{region '#Template'}
	{attribute 'Version' := '5.1.0.1'}
	{attribute 'Tags' := '"LCID": "1031", "Text": "AC, Aggregates, pre-heater, Return temperature control"'}
	{attribute 'Tags' := '"LCID": "1033", "Text": "AC, Aggregates, pre-heater, Return temperature control"'}
	{attribute 'Using' := '"Type": "Template", "URI": "BA2_Param"'}
	{attribute 'Using' := '"Type": "Template", "URI": "EC_ID"'}
	{attribute 'Description' := '"LCID": "1031", "Text": "Vorerhitzer Rücklauf Temperatur Regelung"'}
	{attribute 'Description' := '"LCID": "1033", "Text": "Pre-Heater return temperature control"'}
{endregion}
FUNCTION_BLOCK FB_BA_AC_TRtCtrl EXTENDS FB_BA_View
VAR_INPUT
	bEnPreRinse				: BOOL;
	fTRt					: REAL;
	bTWthLowLimit			: BOOL;// Außentemperatur unterer Grenzwert aktiv
	fTWth					: REAL;
	bSkipPreRinse			: BOOL; // Vorspülen überspringen // Skip pre-rinse
	bSeqActive				: BOOL;// Sequenz Regelung ist aktiv 	
END_VAR
VAR_OUTPUT
	fY						: REAL;
	bPreRinseActive			: BOOL;
	bPreRinseReady			: BOOL;
	bPreRinseDstb			: BOOL;
END_VAR
VAR_INPUT CONSTANT
	SpTRtW					: FB_BA_AV_Op;
	PreRinseDelay			: FB_BA_DlyOn;												 
	PreRinseDst				: FB_BA_BV;													   
	PreRinseSp				: FB_BA_Scale_02;																		
	Ctrl					: FB_BA_Loop;	
END_VAR
VAR
	rtrigPreRinse			: R_TRIG;
	rsPreRinseReady			: RS;
	rsPreRinseActive		: RS;
	PreRinseHys				: FB_BA_Swi2P;
END_VAR

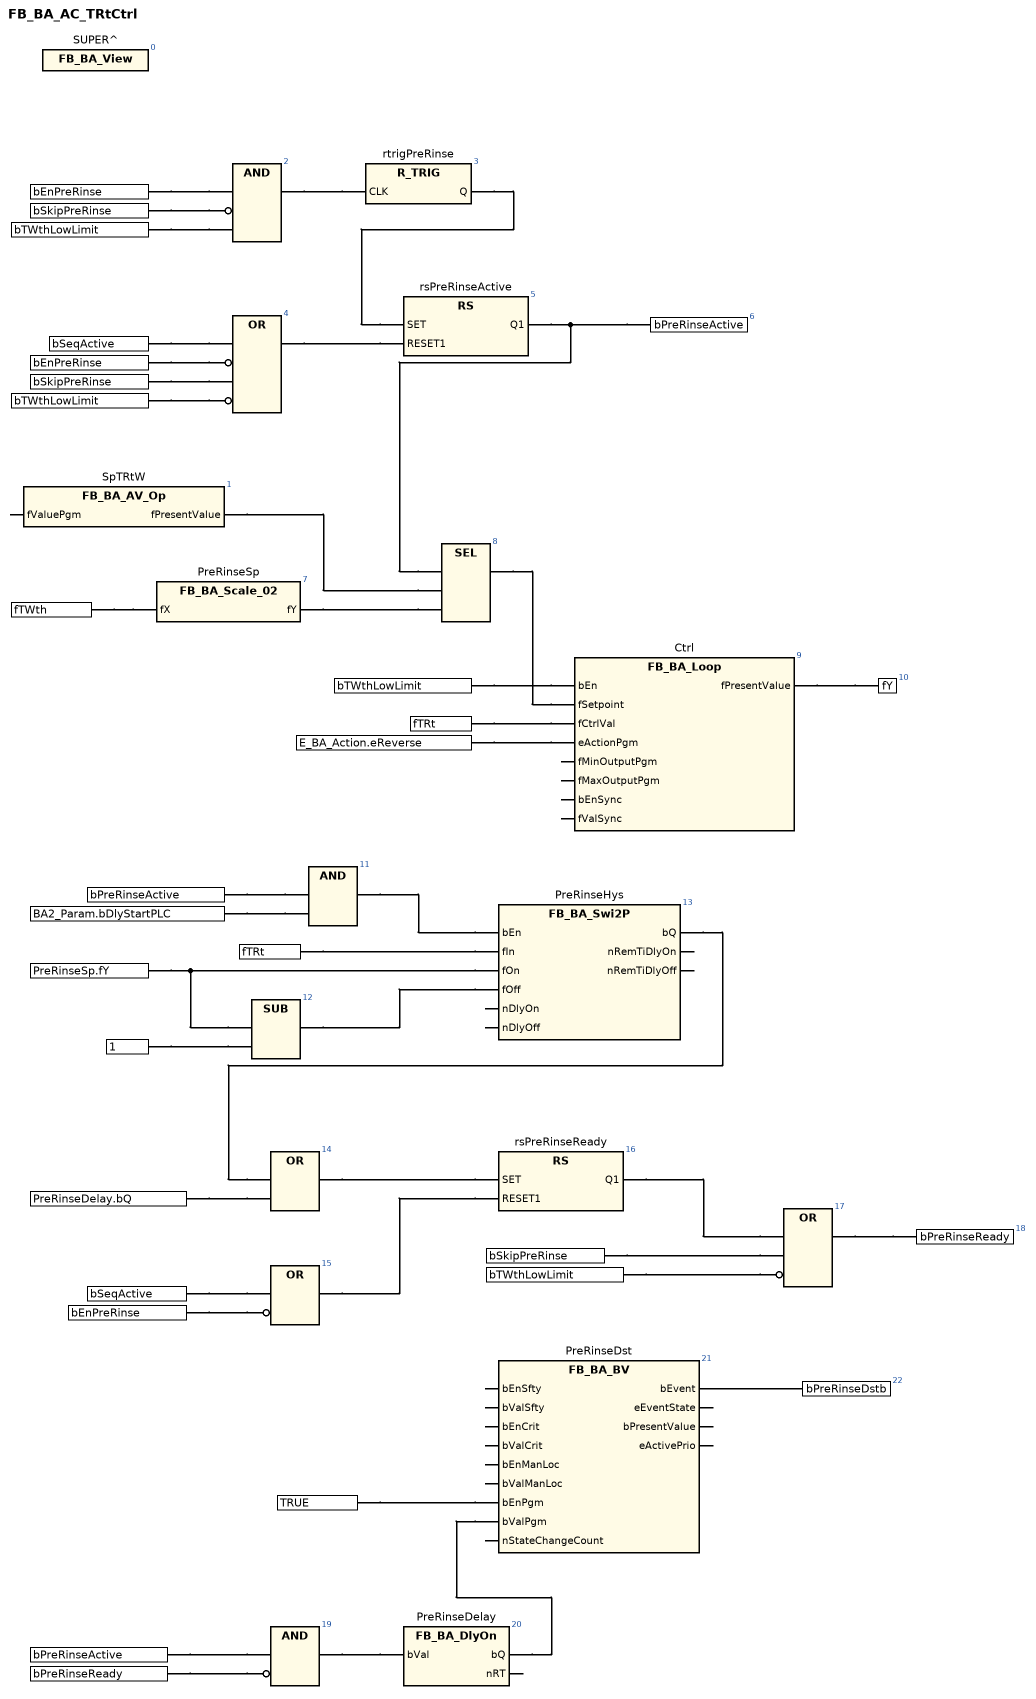
SUPER^(); // FB_BA_View
SpTRtW(); // FB_BA_AV_Op
rtrigPreRinse(CLK := bEnPreRinse AND NOT bSkipPreRinse AND bTWthLowLimit); // R_TRIG
rsPreRinseActive(SET := rtrigPreRinse.Q, RESET1 := bSeqActive OR NOT bEnPreRinse OR bSkipPreRinse OR NOT bTWthLowLimit); // RS
bPreRinseActive := rsPreRinseActive.Q1;
PreRinseSp(fX := fTWth); // FB_BA_Scale_02
Ctrl(
    bEn := bTWthLowLimit,
    fSetpoint := SEL(rsPreRinseActive.Q1, SpTRtW.fPresentValue, PreRinseSp.fY),
    fCtrlVal := fTRt,
    eActionPgm := E_BA_Action.eReverse); // FB_BA_Loop
fY := Ctrl.fPresentValue;
PreRinseHys(
    bEn := bPreRinseActive AND BA2_Param.bDlyStartPLC,
    fIn := fTRt,
    fOn := PreRinseSp.fY,
    fOff := PreRinseSp.fY - 1); // FB_BA_Swi2P
rsPreRinseReady(SET := PreRinseHys.bQ OR PreRinseDelay.bQ, RESET1 := bSeqActive OR NOT bEnPreRinse); // RS
bPreRinseReady := rsPreRinseReady.Q1 OR bSkipPreRinse OR NOT bTWthLowLimit;
PreRinseDelay(bVal := bPreRinseActive AND NOT bPreRinseReady); // FB_BA_DlyOn
PreRinseDst(bEnPgm := TRUE, bValPgm := PreRinseDelay.bQ); // FB_BA_BV
bPreRinseDstb := PreRinseDst.bEvent;

METHOD FB_init : BOOL
VAR_INPUT
	bInitRetains : BOOL; // if TRUE, the retain variables are initialized (warm start / cold start)
	bInCopyCode : BOOL;  // if TRUE, the instance afterwards gets moved into the copy code (online change)
END_VAR
SpTRtW.iParent								:= THIS^;
SpTRtW.iLabel								:= LblFun_Setpoint; 
SpTRtW.sObjectName							:= '{Idx=01}';						 
SpTRtW.eUnit 								:= E_BA_Unit.eTemperature_DegreesCelsius;								 								
SpTRtW.fValueRm								:= 5.0;

PreRinseDelay.iParent						:= THIS^;	
PreRinseDelay.iLabel						:= LblCtl_DelayOn; 
PreRinseDelay.sObjectName					:= '{Idx=01}';						 
PreRinseDelay.eDPADMode						:= E_BA_DPADMode.eIncludeDescription;
PreRinseDelay.TiDly.iLabel					:= LblCtl_PreRinseDuration; 
PreRinseDelay.TiDly.sObjectName				:= '{Idx=01}';						 
PreRinseDelay.TiDly.fValueRm				:= 900;	

PreRinseDst.iParent							:= THIS^;
PreRinseDst.iLabel							:= LblCtl_DisturbancePreRinse; 
PreRinseDst.sObjectName						:= '{Idx=01}';						 
PreRinseDst.bEnOutOfService					:= FALSE;
PreRinseDst.sActiveText 					:= txtEvent_Triggered;
PreRinseDst.sInactiveText 					:= txtEvent_Normal;
PreRinseDst.nStateChangeCount				:= 0;
PreRinseDst.nActiveTimeElapsed				:= 0;
PreRinseDst.nMinimumOnTime					:= 0;
PreRinseDst.nMinimumOffTime					:= 0;
PreRinseDst.bEnManualRm						:= FALSE;	//	Priority  8	
PreRinseDst.bValManualRm					:= FALSE;	//	Priority  8
PreRinseDst.bDefaultValue					:= FALSE;
PreRinseDst.nEventClassID					:= EC_ID.NC30;
PreRinseDst.stTimeDelay.nToNormal			:= 0;
PreRinseDst.stTimeDelay.nToAbnormal			:= 0;
PreRinseDst.bAlarmValue						:= TRUE;
PreRinseDst.bAcknowledgeRm					:= FALSE;		
PreRinseDst.aEventTransitionText[1]			:= txtEvent_Triggered;
PreRinseDst.aEventTransitionText[2]			:= txtEvent_Error;
PreRinseDst.aEventTransitionText[3]			:= txtEvent_Normal;
PreRinseDst.bEventDetectionEnable			:= TRUE;
PreRinseDst.aEventEnable[1]					:= TRUE;			//	to_offnormal
PreRinseDst.aEventEnable[2]					:= FALSE;			//	to_fault
PreRinseDst.aEventEnable[3]					:= TRUE;			//	to_normal
PreRinseDst.eEnPlantLock					:= E_BA_LockPriority.eNoLock;	

PreRinseSp.iParent							:= THIS^;
PreRinseSp.iLabel							:= LblCtl_CalculationPreRinseSetpoint; 
PreRinseSp.sObjectName						:= '{Idx=02}';						 
PreRinseSp.eDPADMode						:= E_BA_DPADMode.eIncludeDescription;
PreRinseSp.X1.fValueRm						:= -10.0;
PreRinseSp.X2.fValueRm						:= 6.0;
PreRinseSp.Y1.fValueRm						:= 30.0;
PreRinseSp.Y2.fValueRm						:= 25.0;
PreRinseSp.YMin.fValueRm					:= 20.0;
PreRinseSp.YMax.fValueRm					:= 60.0;

Ctrl.iParent								:= THIS^;
Ctrl.iLabel									:= LblFun_LoopObject; 
Ctrl.sObjectName							:= '{Idx=01}';						 
Ctrl.eOpMode								:= E_BA_PIDMode.eP1ID;								 	 										 
Ctrl.eOutputUnit							:= E_BA_Unit.eOther_Percent;
Ctrl.eActionRm								:= E_BA_Action.eReverse;
Ctrl.fProportionalConstant					:= 3;
Ctrl.fIntegralConstant						:= 180;
Ctrl.fDerivativeConstant					:= 0;
Ctrl.fMaxOutputRm 							:= 100;
Ctrl.fMinOutputRm							:= 0;
Ctrl.fCOVIncrement							:= 0;
Ctrl.nDampConstant							:= 0;
Ctrl.fNeutralZone							:= 0;
END_METHOD

END_FUNCTION_BLOCK

(* stored: Version 1.1.0.1, ProductVersion 3.1.4024.12
   POU FB_BA_AC_TRtCtrl: Id {ad605d05-9fe2-4df4-883e-9551f7b83caa}, SpecialFunc None
   Method FB_init: Id {a602ee85-f6e5-4f6e-ad67-9f2945317e31} *)
